Staubli VAL3: JointVel.dtx

public num jv1
public num jv2
public num jv3
public num jv4
public num jv5
public num jv6
